// TwinCAT 3 PLC project mobject_commands
// Title: mobject-commands
// Company: mobject
// Author: mobject dev team
// ProjectVersion: 0.1.0
// ProgramVersion: 3.1.4024.0
// libraries:
//   mobject-collections, * (mobject)
//   mobject-disposable, * (mobject)
//   Tc2_System, * (Beckhoff Automation GmbH)
// project tree:
//   AsyncCommand/ DefaultResult.TcPOU, AsyncCommand.TcPOU
//   AsyncCommand/Interface/ I_AsyncCommand.TcIO, I_Result.TcIO
//   AsyncCommand/Runners/ SingleAsyncCommandRunner.TcPOU, QueuedPoolAsyncCommandRunner.TcPOU
//   Command/Interface/ I_Command.TcIO
//   _Internal/AsyncCommandStateMachine/ AsyncCommandStateMachine.TcPOU, I_AsyncCommandStateControl.TcIO
//   _Internal/ CollectionSize.TcDUT

// ---- _Internal/CollectionSize.TcDUT
TYPE CollectionSize : DINT(1..2147483647); END_TYPE

// ---- AsyncCommand/Interface/I_AsyncCommand.TcIO
INTERFACE PUBLIC I_AsyncCommand extends I_Command

METHOD PUBLIC Abort
END_METHOD

METHOD PUBLIC CyclicCall
END_METHOD

{attribute 'monitoring' := 'call'}
PROPERTY PUBLIC Executing : BOOL
GET
END_GET
END_PROPERTY

METHOD PUBLIC GetResult : I_Result
END_METHOD

{attribute 'monitoring' := 'call'}
PROPERTY PUBLIC Idle : BOOL
GET
END_GET
END_PROPERTY

{attribute 'monitoring' := 'call'}
PROPERTY PUBLIC Stopped : BOOL
GET
END_GET
END_PROPERTY

END_INTERFACE

// ---- AsyncCommand/Interface/I_Result.TcIO
INTERFACE I_Result EXTENDS I_Disposable

{attribute 'monitoring' := 'call'}
PROPERTY PUBLIC Aborted : BOOL
GET // PUBLIC
END_GET
END_PROPERTY

{attribute 'monitoring' := 'call'}
PROPERTY PUBLIC Completed : BOOL
GET // PUBLIC
END_GET
END_PROPERTY

{attribute 'monitoring' := 'call'}
PROPERTY PUBLIC Error : BOOL
GET // PUBLIC
END_GET
END_PROPERTY

{attribute 'monitoring' := 'call'}
PROPERTY PUBLIC ErrorId : UDINT
GET // PUBLIC
END_GET
END_PROPERTY

END_INTERFACE

// ---- Command/Interface/I_Command.TcIO
INTERFACE PUBLIC I_Command EXTENDS I_Disposable

METHOD PUBLIC Execute
END_METHOD

END_INTERFACE

// ---- _Internal/AsyncCommandStateMachine/I_AsyncCommandStateControl.TcIO
INTERFACE PUBLIC I_AsyncCommandStateControl

METHOD PUBLIC Error
VAR_INPUT
	errorId : UDINT;
END_VAR
END_METHOD

METHOD PUBLIC Next
END_METHOD

END_INTERFACE

// ---- AsyncCommand/DefaultResult.TcPOU
{attribute 'linkalways'} 
{attribute 'no_explicit_call' := 'This FB is a CLASS and must be accessed using methods or properties'}
{attribute 'enable_dynamic_creation'}
FUNCTION_BLOCK INTERNAL DefaultResult EXTENDS Disposable IMPLEMENTS I_Result
VAR
	_completed : BOOL;
	_aborted : BOOL;
	_error : BOOL;
	_errorId : UDINT;
END_VAR

{attribute 'monitoring' := 'call'}
PROPERTY PUBLIC Aborted : BOOL
GET // PUBLIC
Aborted := _aborted;
END_GET
END_PROPERTY

{attribute 'monitoring' := 'call'}
PROPERTY PUBLIC Completed : BOOL
GET // PUBLIC
Completed := _completed;
END_GET
END_PROPERTY

{attribute 'monitoring' := 'call'}
PROPERTY PUBLIC Error : BOOL
GET // PUBLIC
Error := _error;
END_GET
END_PROPERTY

{attribute 'monitoring' := 'call'}
PROPERTY PUBLIC ErrorId : UDINT
GET // PUBLIC
ErrorId := _errorId;
END_GET
END_PROPERTY

METHOD FB_init : BOOL
VAR_INPUT
	bInitRetains : BOOL; // if TRUE, the retain variables are initialized (warm start / cold start)
	bInCopyCode : BOOL;  // if TRUE, the instance afterwards gets moved into the copy code (online change)
	completed : BOOL;
	aborted : BOOL;
	error : BOOL;
	errorId : UDINT;
END_VAR
THIS^._completed := completed;
THIS^._aborted := aborted;
THIS^._error := error;
THIS^._errorId := errorId;
END_METHOD

END_FUNCTION_BLOCK

// ---- AsyncCommand/AsyncCommand.TcPOU
{attribute 'linkalways'} 
{attribute 'no_explicit_call' := 'This FB is a CLASS and must be accessed using methods or properties'}
{attribute 'enable_dynamic_creation'}
FUNCTION_BLOCK PUBLIC ABSTRACT AsyncCommand EXTENDS Disposable IMPLEMENTS I_AsyncCommand
VAR
	stateMachine : AsyncCommandStateMachine;
END_VAR

(*
 Output   │ Idle     . Executing                                              . Stopped
──────────┼───────────────────────────────────────────────────────────────────────────────────
 State    │          .                                                        .
          │ ┌──────┐ . ┌──────────────┐  ┌───────────┐  ┌────────────┐        . ┌───────────┐
          │ │ Idle ├───► Initializing ├──► Executing ├──► Completing ├──────────► Completed │
          │ └──────┘ . └────┬─────────┘  └────┬──┬───┘  └─────┬──────┘        . └───────────┘
          │          .      │                 │  │            │               .
          │          .      │                 │  │            │  ┌──────────┐ . ┌─────────┐
          │          .      │                 │  └────────────│──► Aborting ├───► Aborted │
          │          .      │                 │               │  └────┬─────┘ . └─────────┘
          │          .      │                 │               │       |       .
          │          .      │                 │               │       │       . ┌──────────┐
          │          .      └─────────────────▼───────────────▼───────▼─────────► Errored  │
          │          .                                                        . └──────────┘
*)

METHOD PUBLIC Abort
stateMachine.Abort();
END_METHOD

METHOD PUBLIC CyclicCall
IF stateMachine.IsIdle THEN
	OnIdle();
END_IF

IF stateMachine.IsInitializing THEN
	OnInitializing(stateMachine);
END_IF

IF stateMachine.IsExecuting THEN
	OnExecuting(stateMachine);
END_IF

IF stateMachine.IsCompleting THEN
	OnCompleting(stateMachine);
END_IF

IF stateMachine.IsCompleted THEN
	OnCompleted();
END_IF

IF stateMachine.IsAborting THEN
	OnAborting(stateMachine);
END_IF

IF stateMachine.IsAborted THEN
	OnAborted();
END_IF

IF stateMachine.IsErrored THEN
	OnErrored();
END_IF
END_METHOD

METHOD PUBLIC Execute
stateMachine.Execute();
END_METHOD

{attribute 'monitoring' := 'call'}
PROPERTY PUBLIC Executing : BOOL
GET // PUBLIC
IF stateMachine.IsAborted THEN
	RETURN;
END_IF

IF stateMachine.IsCompleted THEN
	RETURN;
END_IF

IF stateMachine.IsErrored THEN
	RETURN;
END_IF

IF stateMachine.IsIdle THEN
	RETURN;
END_IF

Executing := TRUE;
END_GET
END_PROPERTY

METHOD PUBLIC GetResult : I_Result
VAR
	pResult : POINTER TO DefaultResult;
END_VAR
IF NOT Stopped THEN
	RETURN;
END_IF

pResult := __NEW(DefaultResult(
	completed := stateMachine.IsCompleted,
	aborted := stateMachine.IsAborted,
	error := stateMachine.IsErrored,
	errorId := stateMachine.ErrorId
));

GetResult := pResult^;
END_METHOD

{attribute 'monitoring' := 'call'}
PROPERTY PUBLIC Idle : BOOL
GET // PUBLIC
Idle := stateMachine.IsIdle;
END_GET
END_PROPERTY

METHOD PROTECTED OnAborted
END_METHOD

METHOD PROTECTED OnAborting
VAR_INPUT
	stateControl : I_AsyncCommandStateControl;
END_VAR
// default behaviour is to go to next state
// you can override this method to implement your own completing control code.
// just call StateControl.Next() when your code is completed.  

stateControl.Next();
END_METHOD

METHOD PROTECTED OnCompleted : BOOL
END_METHOD

METHOD PROTECTED OnCompleting
VAR_INPUT
	stateControl : I_AsyncCommandStateControl;
END_VAR
// default behaviour is to go to next state
// you can override this method to implement your own completing control code.
// just call StateControl.Next() when your code is completed.  

stateControl.Next();
END_METHOD

METHOD PROTECTED OnErrored
END_METHOD

METHOD PROTECTED OnExecuting
VAR_INPUT
	stateControl : I_AsyncCommandStateControl;
END_VAR
// default behaviour is to go to next state
// you can override this method to implement your own executing control code.
// just call StateControl.Next() when your code is completed.  

stateControl.Next();
END_METHOD

METHOD PROTECTED OnIdle
END_METHOD

METHOD PROTECTED OnInitializing
VAR_INPUT
	stateControl : I_AsyncCommandStateControl;
END_VAR
// default behaviour is to go to next state
// you can override this method to implement your own initializing control code.
// just call StateControl.Next() when your code is completed.  

stateControl.Next();
END_METHOD

{attribute 'monitoring' := 'call'}
PROPERTY PUBLIC Stopped : BOOL
GET // PUBLIC
IF stateMachine.IsIdle THEN
	RETURN;
END_IF

IF stateMachine.IsInitializing THEN
	RETURN;
END_IF

IF stateMachine.IsExecuting THEN
	RETURN;
END_IF

IF stateMachine.IsCompleting THEN
	RETURN;
END_IF

IF stateMachine.IsAborting THEN
	RETURN;
END_IF

Stopped := TRUE;
END_GET
END_PROPERTY

END_FUNCTION_BLOCK

// ---- _Internal/AsyncCommandStateMachine/AsyncCommandStateMachine.TcPOU
{attribute 'linkalways'} 
{attribute 'no_explicit_call' := 'This FB is a CLASS and must be accessed using methods or properties'}
{attribute 'enable_dynamic_creation'}
FUNCTION_BLOCK INTERNAL AsyncCommandStateMachine IMPLEMENTS I_AsyncCommandStateControl
VAR
	state : (IDLE, INITIALIZING, EXECUTING, COMPLETING, COMPLETED, ABORTING, ABORTED, ERRORED);
	_errorId : UDINT;
END_VAR

(*
State Machine
    ┌──────┐
    │ Idle │
    └──┬───┘
       │                    Error
       │ Execute           ┌────────────────────────────────────────┐
       │                   │                                        │
┌──────▼───────┐ Next ┌────┴──────┐ Next ┌────────────┐ Error       │
│ Initializing ├──────► Executing ├──────► Completing ├──────────┐  │
└──────┬───────┘      └────┬──────┘      └─────┬──────┘          │  │
       │                   │                   │                 │  │
       │ Error             │ Abort             │ Next            │  │
       │                   │                   │                 │  │
       │              ┌────▼─────┐ Error       │                 │  │
       │              │ Aborting ├─────────────┼──────────────┐  │  │
       │              └────┬─────┘             │              │  │  │
       │                   │                   │              │  │  │
       │                   │ Next              │              │  │  │
       │                   │                   │              │  │  │
       │              ┌────▼────┐        ┌─────▼─────┐      ┌─▼──▼──▼─┐
       │              │ Aborted │        │ Completed │      │ Errored │
       │              └─────────┘        └───────────┘      └────▲────┘
       │                                                         │
       └─────────────────────────────────────────────────────────┘
*)

METHOD PUBLIC Abort
CASE state OF
	IDLE : RETURN;
	ABORTING : RETURN;
	COMPLETED : RETURN;
	ABORTED : RETURN;
	ERRORED : RETURN;
END_CASE

state := ABORTING;
END_METHOD

METHOD PUBLIC Error
VAR_INPUT
	errorId : UDINT;
END_VAR
CASE state OF
	IDLE : RETURN;
	COMPLETED : RETURN;
	ABORTED : RETURN;
	ERRORED : RETURN;
END_CASE

_errorId := errorId;
state := ERRORED;
END_METHOD

{attribute 'monitoring' := 'call'}
PROPERTY PUBLIC ErrorId : UDINT
GET // PUBLIC
ErrorId := _errorId;
END_GET
END_PROPERTY

METHOD PUBLIC Execute
CASE state OF
	INITIALIZING : RETURN;
	EXECUTING : RETURN;
	COMPLETING : RETURN;
	ABORTING : RETURN;
END_CASE

_errorId := 0;
state := INITIALIZING;
END_METHOD

{attribute 'monitoring' := 'call'}
PROPERTY PUBLIC IsAborted : BOOL
GET // PUBLIC
IsAborted := state = ABORTED;
END_GET
END_PROPERTY

{attribute 'monitoring' := 'call'}
PROPERTY PUBLIC IsAborting : BOOL
GET // PUBLIC
IsAborting := state = ABORTING;
END_GET
END_PROPERTY

{attribute 'monitoring' := 'call'}
PROPERTY PUBLIC IsCompleted : BOOL
GET // PUBLIC
IsCompleted := state = COMPLETED;
END_GET
END_PROPERTY

{attribute 'monitoring' := 'call'}
PROPERTY PUBLIC IsCompleting : BOOL
GET // PUBLIC
IsCompleting := state = COMPLETING;
END_GET
END_PROPERTY

{attribute 'monitoring' := 'call'}
PROPERTY PUBLIC IsErrored : BOOL
GET // PUBLIC
IsErrored := state = ERRORED;
END_GET
END_PROPERTY

{attribute 'monitoring' := 'call'}
PROPERTY PUBLIC IsExecuting : BOOL
GET // PUBLIC
IsExecuting := state = EXECUTING;
END_GET
END_PROPERTY

{attribute 'monitoring' := 'call'}
PROPERTY PUBLIC IsIdle : BOOL
GET // PUBLIC
IsIdle:= state = IDLE;
END_GET
END_PROPERTY

{attribute 'monitoring' := 'call'}
PROPERTY PUBLIC IsInitializing : BOOL
GET // PUBLIC
IsInitializing := state = INITIALIZING;
END_GET
END_PROPERTY

METHOD PUBLIC Next
CASE state OF
	IDLE : RETURN;
	INITIALIZING : StateComplete_Initializing();
	EXECUTING : StateComplete_Executing();
	COMPLETING : StateComplete_Completing();
	COMPLETED : RETURN;
	ABORTING : StateComplete_Aborting();
	ABORTED : RETURN;
	ERRORED : RETURN;
END_CASE
END_METHOD

METHOD PRIVATE StateComplete_Aborting
state := ABORTED;
END_METHOD

METHOD PRIVATE StateComplete_Completing
state := COMPLETED;
END_METHOD

METHOD PRIVATE StateComplete_Executing
state := COMPLETING;
END_METHOD

METHOD PRIVATE StateComplete_Initializing
state := EXECUTING;
END_METHOD

END_FUNCTION_BLOCK

// ---- AsyncCommand/Runners/SingleAsyncCommandRunner.TcPOU
{attribute 'linkalways'} 
{attribute 'no_explicit_call' := 'This FB is a CLASS and must be accessed using methods or properties'}
{attribute 'enable_dynamic_creation'}
FUNCTION_BLOCK SingleAsyncCommandRunner
VAR
	currentCommand : I_AsyncCommand;
	replacementCommand : I_AsyncCommand;
END_VAR

METHOD PUBLIC CyclicCall
IF currentCommand <> 0 AND_THEN NOT currentCommand.Idle THEN
	currentCommand.CyclicCall();
	RETURN;
END_IF

IF replacementCommand <> 0 THEN
	currentCommand := replacementCommand;
	replacementCommand := 0;
	currentCommand.Execute();
END_IF
END_METHOD

METHOD ExecuteCommand
VAR_INPUT
	Command : I_AsyncCommand;
END_VAR
IF currentCommand = 0 THEN
	currentCommand := Command;
	currentCommand.Execute();
	RETURN;
END_IF

currentCommand.Abort();
replacementCommand := Command;
END_METHOD

{attribute 'monitoring' := 'call'}
PROPERTY PUBLIC Executing : BOOL
GET // PUBLIC
IF currentCommand = 0 THEN
	RETURN;
END_IF

Executing := currentCommand.Executing;
END_GET
END_PROPERTY

METHOD PUBLIC GetResult : I_Result
IF currentCommand = 0 THEN
	RETURN;
END_IF

GetResult := currentCommand.GetResult();
END_METHOD

{attribute 'monitoring' := 'call'}
PROPERTY PUBLIC Idle : BOOL
GET // PUBLIC
IF currentCommand = 0 THEN
	RETURN;
END_IF

Idle := currentCommand.Idle;
END_GET
END_PROPERTY

{attribute 'monitoring' := 'call'}
PROPERTY PUBLIC Stopped : BOOL
GET // PUBLIC
IF currentCommand = 0 THEN
	RETURN;
END_IF

Stopped := currentCommand.Stopped;
END_GET
END_PROPERTY

END_FUNCTION_BLOCK

// ---- AsyncCommand/Runners/QueuedPoolAsyncCommandRunner.TcPOU
{attribute 'linkalways'} 
{attribute 'no_explicit_call' := 'This FB is a CLASS and must be accessed using methods or properties'}
{attribute 'enable_dynamic_creation'}
FUNCTION_BLOCK QueuedPoolAsyncCommandRunner
VAR
	pool : LinkedList;
	queue : Queue;
	poolCapacity : CollectionSize;
	queueCapacity : CollectionSize;
END_VAR

METHOD PUBLIC CyclicCall
VAR
	enumerator : mobject_collections.I_ForwardEnumerator;
	command : I_AsyncCommand;
END_VAR
IF pool.Count < poolCapacity THEN
	// Need to think about how we handle errors
	IF queue.TryDequeue(command) THEN
		pool.AddLast(command);
		command.Execute();
	END_IF
END_IF

IF pool.Count > 0 THEN
	enumerator := pool.GetEnumerator();
	WHILE enumerator.MoveNext() DO
		IF enumerator.TryGet(command) THEN
			IF command <> 0 THEN
				IF command.Idle THEN
					command.Execute();
				ELSIF command.Executing THEN
					command.CyclicCall();
				ELSIF command.Stopped THEN
					pool.Remove(command);
				END_IF
			END_IF
		END_IF
	END_WHILE
	enumerator.Dispose();
END_IF
END_METHOD

METHOD FB_init : BOOL
VAR_INPUT
	bInitRetains : BOOL; // if TRUE, the retain variables are initialized (warm start / cold start)
	bInCopyCode : BOOL;  // if TRUE, the instance afterwards gets moved into the copy code (online change)
	poolCapacity : CollectionSize; // DINT(1..2147483647)
	queueCapacity : CollectionSize;
END_VAR
THIS^.poolCapacity := poolCapacity;
THIS^.queueCapacity := queueCapacity;
END_METHOD

{attribute 'monitoring' := 'call'}
PROPERTY PUBLIC PoolCount : DINT
GET // PUBLIC
PoolCount := pool.Count;
END_GET
END_PROPERTY

METHOD PUBLIC QueueCommand : BOOL
VAR_INPUT
	command : I_AsyncCommand;
END_VAR
IF pool.Count < poolCapacity THEN
	pool.AddLast(command);
	QueueCommand := TRUE;
	RETURN;
END_IF

IF queue.Count < queueCapacity THEN
	queue.Enqueue(command);
	QueueCommand := TRUE;
	RETURN;
END_IF
END_METHOD

{attribute 'monitoring' := 'call'}
PROPERTY PUBLIC QueueCount : DINT
GET // PUBLIC
QueueCount := queue.Count;
END_GET
END_PROPERTY

END_FUNCTION_BLOCK
